// TIA Portal V20 export
DATA_BLOCK "LPFE_TxnBuffer"   // DB250
TITLE = Buffer of RequestOrderInfo messages
// Contains acknowledged transactions until combined to a txn message
// stored: Access Published, MemoryReserve 100, Namespace PFE
   VAR
      buffer { ExternalAccessible := 'False'; ExternalVisible := 'False'; ExternalWritable := 'False'} : Array[0.._.NUMBER_TXN_PER_MESSAGE] of "LPFE_typePFEData";   // Buffer where txn are collected
      mgmtBuffer { ExternalAccessible := 'False'; ExternalVisible := 'False'; ExternalWritable := 'False'} : "LPFE_typeMsgBuffer";   // Management struct of buffer where txn are collected
   END_VAR
BEGIN
END_DATA_BLOCK
